(* CODESYS project chaincontroller_3028.library
   Author: Filippo Boido
   Placeholder: ChainControllerLib
   Title: ChainControllerLib
   Version: 3.0.2.8
   DocFormat: reStructuredText
   Company: FactoryAutomation

Project tree, tasks and I/O mapping:
  libraries: StateMachineLib, * (FactoryAutomation); StepWorkerLib, * (FactoryAutomation); Tc2_Standard, * (Beckhoff Automation GmbH); Tc2_System, * (Beckhoff Automation GmbH); Tc3_Module, * (Beckhoff Automation GmbH)
  DUTs/
    data type ST_ChainDefinition
    data type ST_ChainStateMachine
  GVLs/
    global variables GVL_Constants
  POUs/
    function block FB_Chain [ST]: getDefinition, getRefChainReleases, getRefReleaseResult, getReleaseResult
    function block FB_ChainController [ST]: addChain, releaseCheck, releaseForChain, releaseFromChain, releaseResult
    function block FB_TestChain1 [ST]: Busy, Error, Idle, Init, Prepare, Ready, Waiting
    function block FB_TestChain2 [ST]: Busy, Error, Idle, Init, Prepare, Ready, Waiting
    interface I_Chain: getDefinition, getRefChainReleases, getRefReleaseResult
    interface I_ChainController: addChain, releaseForChain, releaseFromChain, releaseResult
    program MAIN [ST]
  VISUs/
  program Version [ST]
*)

// DUTs/ST_ChainDefinition
TYPE ST_ChainDefinition :
STRUCT
	uiChainNumber : UINT;
	sChainName : STRING;
END_STRUCT
END_TYPE

// DUTs/ST_ChainStateMachine
TYPE ST_ChainStateMachine :
STRUCT
	bInit : BOOL;
	bReady : BOOL;
	bBusy : BOOL;
	bStop : BOOL;
	bWait : BOOL;
	bError : BOOL;
END_STRUCT
END_TYPE

// GVLs/GVL_Constants

VAR_GLOBAL CONSTANT
	cMaxChains : UINT := 50;
END_VAR

// POUs/FB_Chain
FUNCTION_BLOCK ABSTRACT FB_Chain EXTENDS StateMachine IMPLEMENTS I_Chain
VAR_INPUT CONSTANT
	uiChainNumber : UINT;
	sChainName : STRING;
	rChainController : REFERENCE TO FB_ChainController;
END_VAR

VAR_OUTPUT
	bReleaseResult : BOOL;
END_VAR
VAR

	fbReleaseResult : BoolOut;
	aChainReleases : ARRAY[1..cMaxChains] OF BOOL;

	fbStepWorkerInit : FB_StepWorker;
	fbStepWorkerReady : FB_StepWorker;
	fbStepWorkerBusy : FB_StepWorker;
	fbStepWorkerWaiting : FB_StepWorker;
	fbStepWorkerError : FB_StepWorker;

END_VAR

IF sChainName = '' 
	OR NOT __ISVALIDREF(rChainController)
THEN
	
	eStateMachine := eError;
	RETURN;
END_IF

SUPER^();
bReleaseResult := fbReleaseResult.getValue;

PROPERTY getDefinition : ST_ChainDefinition
GET
getDefinition.sChainName := sChainName;
getDefinition.uiChainNumber := uiChainNumber;
END_GET
END_PROPERTY

PROPERTY getRefChainReleases : REFERENCE TO ARRAY[1..cMaxChains] OF BOOL
GET
getRefChainReleases REF= aChainReleases;
END_GET
END_PROPERTY

{warning 'Eigenschaftenimplementierung hinzufügen'}
PROPERTY getRefReleaseResult : REFERENCE TO BOOL
GET
getRefReleaseResult REF= bReleaseResult;
END_GET
END_PROPERTY

PROPERTY getReleaseResult : BoolOut
GET
getReleaseResult := fbReleaseResult;
END_GET
END_PROPERTY

END_FUNCTION_BLOCK

// POUs/I_Chain
INTERFACE I_Chain

PROPERTY getDefinition : ST_ChainDefinition
GET
END_GET
END_PROPERTY

PROPERTY getRefChainReleases : REFERENCE TO ARRAY[1..cMaxChains] OF BOOL
GET
END_GET
END_PROPERTY

PROPERTY getRefReleaseResult : REFERENCE TO BOOL
GET
END_GET
END_PROPERTY

END_INTERFACE

// POUs/FB_ChainController
{attribute 'enable_dynamic_creation'}
FUNCTION_BLOCK FB_ChainController IMPLEMENTS I_ChainController
VAR_INPUT
	
END_VAR
VAR_OUTPUT
END_VAR
VAR
	aChains : ARRAY[1..cMaxChains] OF I_Chain;
	uiNextChain : UINT := 1;
END_VAR

METHOD addChain : I_ChainController 
VAR_INPUT
	itfChain : I_Chain;
END_VAR
VAR
	i: UINT;
END_VAR
addChain := THIS^;

IF itfChain = 0 
OR uiNextChain > cMaxChains 
THEN
	RETURN;
END_IF

//chain already added?
FOR i := 1 TO uiNextChain-1 DO
	IF aChains[i] = itfChain
	THEN
		//yes, already added
		RETURN;
	END_IF
END_FOR

aChains[uiNextChain] := itfChain;
uiNextChain := uiNextChain + 1;
END_METHOD

METHOD releaseCheck : I_ChainController
VAR_INPUT
	itfContractor : I_Chain;
END_VAR
VAR
	i : UINT;
	rReleaseResult :  REFERENCE TO BOOL; 
END_VAR
releaseCheck := THIS^;

FOR i := 1 TO uiNextChain-1 DO
	
	IF itfContractor = aChains[i]
	THEN
		
		rReleaseResult REF= aChains[i].getRefReleaseResult;
		rReleaseResult := TRUE;
		EXIT;
	END_IF
	
END_FOR
END_METHOD

METHOD Public releaseForChain : I_ChainController
VAR_INPUT
	sChainToRelease : STRING;
	itfCommissioner : I_Chain;
END_VAR
VAR
	i : UINT;
	j: UINT;
	stChainDefinition : ST_ChainDefinition; 
	aChainReleases : REFERENCE TO ARRAY[1..cMaxChains] OF BOOL;
END_VAR
releaseForChain := THIS^;

//search for the chain to release
FOR i := 1 TO uiNextChain-1 DO
	stChainDefinition := aChains[i].GetDefinition;
	IF  stChainDefinition.sChainName = sChainToRelease
	THEN
		aChainReleases REF= aChains[i].getRefChainReleases;
		//search for the commissioner
		FOR j := 1 TO uiNextChain-1 DO
			IF aChains[j] = itfCommissioner
			THEN
				aChainReleases[j] := TRUE;
			END_IF
		END_FOR
			
	END_IF
END_FOR
END_METHOD

METHOD Public releaseFromChain : I_ChainController
VAR_INPUT
	sChainReleasing : STRING;
	itfContractor : I_Chain;
END_VAR
VAR
	i : UINT;
	j: UINT;
	stChainDefinition : ST_ChainDefinition; 
	aChainReleases : REFERENCE TO ARRAY[1..cMaxChains] OF BOOL;
	rReleaseResult : REFERENCE TO BOOL; 
END_VAR
releaseFromChain := THIS^;

//search for the contractor
FOR i := 1 TO uiNextChain-1 DO
	
	IF itfContractor = aChains[i]
	THEN
		aChainReleases REF= aChains[i].getRefChainReleases;
		rReleaseResult REF= aChains[i].getRefReleaseResult;
		FOR j := 1 TO uiNextChain-1 DO
			stChainDefinition := aChains[j].getDefinition;
			IF stChainDefinition.sChainName = sChainReleasing
			THEN
				rReleaseResult := rReleaseResult AND aChainReleases[j]; 
			END_IF
			
		END_FOR
		
	END_IF
	
END_FOR
END_METHOD

METHOD releaseResult : Bool
VAR_INPUT
	itfRequester : I_Chain;
END_VAR
VAR
	i,j : UINT;
	rReleaseResult : REFERENCE TO BOOL; 
	aChainReleases : REFERENCE TO ARRAY[1..cMaxChains] OF BOOL;
END_VAR
FOR i := 1 TO cMaxChains DO
	
	IF  itfRequester = aChains[i]
	THEN
		IF aChains[i].getRefReleaseResult 
		THEN
			releaseResult := TRUE;
			aChainReleases REF= aChains[i].getRefChainReleases;
			//reset the releases
			FOR j := 1 TO uiNextChain-1 DO
				aChainReleases[j] := FALSE;
			END_FOR
			EXIT;
		END_IF
	END_IF
END_FOR
END_METHOD

END_FUNCTION_BLOCK

// POUs/I_ChainController
INTERFACE I_ChainController

METHOD addChain : I_ChainController 
VAR_INPUT
	itfChain : I_Chain;
END_VAR
END_METHOD

METHOD releaseForChain : I_ChainController
VAR_INPUT
	sChainToRelease : STRING;
	itfCommissioner : I_Chain;
END_VAR
END_METHOD

METHOD releaseFromChain : I_ChainController
VAR_INPUT
	sChainReleasing : STRING;
	itfContractor : I_Chain;
END_VAR
END_METHOD

METHOD releaseResult : Bool
VAR_INPUT
	itfRequester : I_Chain;
END_VAR
END_METHOD

END_INTERFACE

// POUs/FB_TestChain1
FUNCTION_BLOCK FB_TestChain1 EXTENDS FB_Chain
VAR_INPUT
END_VAR
VAR_OUTPUT
END_VAR
VAR
END_VAR

super^();

METHOD PROTECTED Busy : BOOL
VAR_INPUT
END_VAR
CASE fbStepWorkerBusy.uiStep OF

0:
	;
10:
	IF rChainController
		.releaseCheck(THIS^)
		.releaseFromChain(sChainReleasing := 'fbChain2', THIS^)
		.releaseResult(THIS^) 
	THEN
		fbStepWorkerBusy.mNextStep(20);
	END_IF
20:
	;
30:

END_CASE
END_METHOD

METHOD PROTECTED Error : BOOL
VAR_INPUT
END_VAR
END_METHOD

METHOD PROTECTED Idle : BOOL
VAR_INPUT
END_VAR
END_METHOD

METHOD PROTECTED Init : BOOL
VAR_INPUT
END_VAR
Start();
END_METHOD

METHOD PROTECTED Prepare : BOOL
VAR_INPUT
END_VAR
END_METHOD

METHOD PROTECTED Ready : BOOL
VAR_INPUT
END_VAR
END_METHOD

METHOD PROTECTED Waiting : BOOL
VAR_INPUT
END_VAR
END_METHOD

END_FUNCTION_BLOCK

// POUs/FB_TestChain2
FUNCTION_BLOCK FB_TestChain2 EXTENDS FB_Chain
VAR_INPUT
END_VAR
VAR_OUTPUT
END_VAR
VAR
END_VAR

super^();

METHOD PROTECTED Busy : BOOL
VAR_INPUT
END_VAR
CASE fbStepWorkerBusy.uiStep OF
0:

10:
	rChainController.releaseForChain(sChainToRelease := 'fbChain1',THIS^);
	fbStepWorkerBusy.mNextStep(20);
20:

30:

END_CASE
END_METHOD

METHOD PROTECTED Error : BOOL
VAR_INPUT
END_VAR
END_METHOD

METHOD PROTECTED Idle : BOOL
VAR_INPUT
END_VAR
END_METHOD

METHOD PROTECTED Init : BOOL
VAR_INPUT
END_VAR
Start();
END_METHOD

METHOD PROTECTED Prepare : BOOL
VAR_INPUT
END_VAR
END_METHOD

METHOD PROTECTED Ready : BOOL
VAR_INPUT
END_VAR
END_METHOD

METHOD PROTECTED Waiting : BOOL
VAR_INPUT
END_VAR
END_METHOD

END_FUNCTION_BLOCK

// POUs/MAIN
PROGRAM MAIN
VAR
	step : UINT;
	fbChainController : FB_ChainController;
	fbChain1 : 	FB_TestChain1 := (sChainName :='fbChain',rChainController :=fbChainController);
	fbChain2 : FB_TestChain2 := (sChainName:='fbChain',rChainController:=fbChainController);
END_VAR

fbChain1();
fbChain2();


CASE step OF

	10: 
		
		fbChainController
			.addChain(fbChain1)
			.addChain(fbChain2);
		
		fbChain1.Execute();
		fbChain2.Execute();	
		step := 20;
		
	20:
	
		
END_CASE

END_PROGRAM

// Version
PROGRAM Version
VAR
END_VAR

(*
1.1.0.1:	Boido	010120

Added new versioning System.
To update the project version open the VersionLib and modify the parameters.

1.1.1.2:	Boido	010120

Deleted the var_io chaincontroller from FB_Chain.
ChainController must now be set with the help of the define method in FB_Chain.

2.0.0.3:	Boido	010120

Deleted the define method from FB_Chain.
Initialization of FB_Chain occurs through FB_init in FB_Chain

2.0.1.4:	Boido	020120

Version.txt replaced with Version PRG

2.0.2.5:	Boido	020120

VersionLib removed.

3.0.0.6:	Boido	020120

FB_init removed from FB_Chain.

3.0.1.7:	Boido 	040120

Removed callAfterInit method from FB_Chain
Check for null reference in FB_Chain

3.0.2.8:	Boido 	050120

E_ChainStateMachine deleted.
*)

END_PROGRAM
